TYPE ST_Position :
STRUCT
	Xpos: REAL;
	Ypos: REAL;
	Zpos: REAL;
	Apos: REAL;
END_STRUCT
END_TYPE

(* stored: Version 1.1.0.1, ProductVersion 3.1.4024.11
   DUT ST_Position: Id {fb0e1fc1-1d22-4bd4-ab81-b4554f59babc} *)
